INTERFACE ITF_LinkedList

METHOD CreateNode : BOOL
END_METHOD

METHOD DestroyNode : BOOL
VAR_INPUT
	Index		: UINT;
END_VAR
END_METHOD

METHOD GetListLength : UINT
VAR_INPUT
END_VAR
END_METHOD

METHOD GetNode : ITF_Node
VAR_INPUT
	Index	: UINT;
END_VAR
END_METHOD

END_INTERFACE

(* stored: Version 1.1.0.1
   Itf ITF_LinkedList: Id {29ba7d83-d588-4c91-a07a-ac71bb854e67}
   Method CreateNode: Id {7316e16a-9a25-4a9f-8d84-207735dd7ed5}
   Method DestroyNode: Id {01e5e783-b54e-4c86-8226-42249c0a8a75}
   Method GetListLength: Id {39ad9b36-39f6-4720-97d9-c6079edb8b99}
   Method GetNode: Id {2ec29a15-c236-42bf-92d3-64ec2951ff5e} *)
